(* IEC 61131-3 sources: ST_L/Practice/02_Control, 5 files *)

(* ---- 02_01_IFDemo.st ---- *)
(* ============================================================================
 * 文件: 02_01_IFDemo.st
 * 章节: 第4章 - 条件控制语句
 * 描述: IF语句完整演示
 * 学习目标: 掌握IF条件语句的各种用法
 * ============================================================================ *)

PROGRAM IFDemo
VAR
    // ==========================================================================
    // 温度监控变量
    // ==========================================================================
    iTemperature : INT := 75;      // 当前温度
    iHighLimit : INT := 100;       // 高温限值
    iLowLimit : INT := 20;         // 低温限值
    iWarningLimit : INT := 80;     // 警告限值
    bHighAlarm : BOOL;             // 高温报警
    bLowAlarm : BOOL;              // 低温报警
    bWarning : BOOL;               // 警告状态

    // ==========================================================================
    // 电机控制变量
    // ==========================================================================
    iMotorSpeed : INT := 0;
    iTargetSpeed : INT := 1500;
    bMotorRunning : BOOL := FALSE;
    bStartButton : BOOL := TRUE;
    bStopButton : BOOL := FALSE;
    bEmergencyStop : BOOL := FALSE;

    // ==========================================================================
    // 数值判断变量
    // ==========================================================================
    iScore : INT := 85;
    sGrade : STRING(2);

    iValue1, iValue2 : INT := 10;
    iMax, iMin, iMid : INT;

    // ==========================================================================
    // 边沿检测变量
    // ==========================================================================
    bCurrentInput : BOOL := FALSE;
    bLastInput : BOOL := FALSE;
    bRisingEdge : BOOL;
    iEdgeCount : INT := 0;

    // ==========================================================================
    // 数值计算变量
    // ==========================================================================
    rNumber : REAL := -3.7;
    iIntegerPart : INT;
    rFractionalPart : REAL;

    iCounter : INT := 0;
END_VAR

// ============================================================================
// 主程序逻辑
// ============================================================================
BEGIN
    // ==========================================================================
    // 1. 简单IF语句
    // ==========================================================================

    // 如果温度超过100度，触发高温报警
    IF iTemperature > iHighLimit THEN
        bHighAlarm := TRUE;
    END_IF

    // ==========================================================================
    // 2. IF-ELSE双分支
    // ==========================================================================

    // 判断电机运行状态
    IF bMotorRunning THEN
        iMotorSpeed := iTargetSpeed;
    ELSE
        iMotorSpeed := 0;
    END_IF

    // ==========================================================================
    // 3. IF-ELSIF-ELSE多分支 - 温度状态判断
    // ==========================================================================

    // 重置报警状态
    bHighAlarm := FALSE;
    bLowAlarm := FALSE;
    bWarning := FALSE;

    IF iTemperature >= iHighLimit THEN
        bHighAlarm := TRUE;
        bWarning := TRUE;
    ELSIF iTemperature <= iLowLimit THEN
        bLowAlarm := TRUE;
        bWarning := TRUE;
    ELSIF iTemperature >= iWarningLimit THEN
        bWarning := TRUE;
    ELSE
        // 温度正常
        bHighAlarm := FALSE;
        bLowAlarm := FALSE;
        bWarning := FALSE;
    END_IF

    // ==========================================================================
    // 4. IF-ELSIF-ELSE多分支 - 分数等级判定
    // ==========================================================================

    IF iScore >= 90 THEN
        sGrade := 'A';
    ELSIF iScore >= 80 THEN
        sGrade := 'B';
    ELSIF iScore >= 70 THEN
        sGrade := 'C';
    ELSIF iScore >= 60 THEN
        sGrade := 'D';
    ELSE
        sGrade := 'F';
    END_IF

    // ==========================================================================
    // 5. 嵌套IF语句 - 三角形类型判断
    // ==========================================================================
    VAR
        a, b, c : INT := 3;
        sTriangleType : STRING(20);
    END_VAR

    IF a + b > c AND b + c > a AND a + c > b THEN
        IF a = b AND b = c THEN
            sTriangleType := '等边三角形';
        ELSIF a = b OR b = c OR a = c THEN
            sTriangleType := '等腰三角形';
        ELSIF (a * a + b * b = c * c) OR (a * a + c * c = b * b) OR (b * b + c * c = a * a) THEN
            sTriangleType := '直角三角形';
        ELSE
            sTriangleType := '普通三角形';
        END_IF
    ELSE
        sTriangleType := '不能构成三角形';
    END_IF

    // ==========================================================================
    // 6. 求三个数的最大、最小、中间值
    // ==========================================================================

    iValue1 := 30;
    iValue2 := 50;

    VAR iValue3 : INT := 40; END_VAR

    IF iValue1 >= iValue2 THEN
        IF iValue1 >= iValue3 THEN
            iMax := iValue1;
            IF iValue2 >= iValue3 THEN
                iMid := iValue2;
                iMin := iValue3;
            ELSE
                iMid := iValue3;
                iMin := iValue2;
            END_IF
        ELSE
            iMax := iValue3;
            iMid := iValue1;
            iMin := iValue2;
        END_IF
    ELSE
        IF iValue2 >= iValue3 THEN
            iMax := iValue2;
            IF iValue1 >= iValue3 THEN
                iMid := iValue1;
                iMin := iValue3;
            ELSE
                iMid := iValue3;
                iMin := iValue1;
            END_IF
        ELSE
            iMax := iValue3;
            iMid := iValue2;
            iMin := iValue1;
        END_IF
    END_IF

    // ==========================================================================
    // 7. 边沿检测 - 上升沿识别
    // ==========================================================================

    bRisingEdge := bCurrentInput AND NOT bLastInput;

    IF bRisingEdge THEN
        iEdgeCount := iEdgeCount + 1;
    END_IF

    bLastInput := bCurrentInput;

    // ==========================================================================
    // 8. 浮点数处理 - 分离整数和小数部分
    // ==========================================================================

    rNumber := -3.14159;

    IF rNumber < 0.0 THEN
        iIntegerPart := REAL_TO_INT(rNumber) - 1;
    ELSE
        iIntegerPart := REAL_TO_INT(rNumber);
    END_IF

    rFractionalPart := rNumber - INT_TO_REAL(iIntegerPart);

    // ==========================================================================
    // 9. 电机启停控制（综合示例）
    // ==========================================================================

    // 急停优先级最高
    IF bEmergencyStop THEN
        bMotorRunning := FALSE;
        iMotorSpeed := 0;
    ELSIF bStopButton THEN
        bMotorRunning := FALSE;
        iMotorSpeed := 0;
    ELSIF bStartButton THEN
        bMotorRunning := TRUE;
        iMotorSpeed := iTargetSpeed;
    END_IF

    // ==========================================================================
    // 10. 计数器限幅
    // ==========================================================================

    iCounter := iCounter + 1;

    IF iCounter > 1000 THEN
        iCounter := 0;
    END_IF

END_PROGRAM

(* ---- 02_02_CASEDemo.st ---- *)
(* ============================================================================
 * 文件: 02_02_CASEDemo.st
 * 章节: 第4章 - 条件控制语句
 * 描述: CASE语句完整演示
 * 学习目标: 掌握CASE选择语句的各种用法
 * ============================================================================ *)

PROGRAM CASEDemo
VAR
    // ==========================================================================
    // 状态机变量
    // ==========================================================================
    iState : INT := 0;
    sStateName : STRING(30);

    // ==========================================================================
    // 月份处理变量
    // ==========================================================================
    iMonth : INT := 3;
    iDays : INT;
    sMonthName : STRING(20);

    // ==========================================================================
    // 菜单选择变量
    // ==========================================================================
    iMenuSelection : INT := 2;
    bExecute : BOOL := TRUE;

    // ==========================================================================
    // 报警级别变量
    // ==========================================================================
    iAlarmLevel : INT := 2;
    sAlarmMessage : STRING(50);
    bAlarmActive : BOOL := TRUE;

    // ==========================================================================
    // 枚举定义（需要定义在TYPE区域，这里用INT模拟）
    // ==========================================================================
    // MachineState: 0=IDLE, 1=STARTING, 2=RUNNING, 3=STOPPING, 4=FAULT
    iMachineState : INT := 0;

    // ==========================================================================
    // 数值范围变量
    // ==========================================================================
    iScore : INT := 78;
    iGradeLevel : INT;

    // ==========================================================================
    // 命令处理变量
    // ==========================================================================
    iCommand : INT := 16#05;
    bSuccess : BOOL;

    // ==========================================================================
    // 临时变量
    // ==========================================================================
    i : INT;
END_VAR

// ============================================================================
// 主程序逻辑
// ============================================================================
BEGIN
    // ==========================================================================
    // 1. 简单CASE语句 - 状态名称显示
    // ==========================================================================

    iState := 2;  // 假设当前状态为2

    CASE iState OF
        0:  sStateName := '初始化';
        1:  sStateName := '就绪';
        2:  sStateName := '运行中';
        3:  sStateName := '暂停';
        4:  sStateName := '停止';
        5:  sStateName := '故障';
    ELSE
        sStateName := '未知状态';
    END_CASE

    // ==========================================================================
    // 2. CASE语句 - 月份天数判断
    // ==========================================================================

    iMonth := 2;  // 2月

    CASE iMonth OF
        1, 3, 5, 7, 8, 10, 12:   // 大月
            iDays := 31;
        4, 6, 9, 11:               // 小月
            iDays := 30;
        2:                          // 2月
            iDays := 28;           // 假设非闰年
    ELSE
        iDays := 0;
    END_CASE

    // ==========================================================================
    // 3. CASE语句 - 月份名称
    // ==========================================================================

    CASE iMonth OF
        1:  sMonthName := '一月';
        2:  sMonthName := '二月';
        3:  sMonthName := '三月';
        4:  sMonthName := '四月';
        5:  sMonthName := '五月';
        6:  sMonthName := '六月';
        7:  sMonthName := '七月';
        8:  sMonthName := '八月';
        9:  sMonthName := '九月';
        10: sMonthName := '十月';
        11: sMonthName := '十一月';
        12: sMonthName := '十二月';
    ELSE
        sMonthName := '无效月份';
    END_CASE

    // ==========================================================================
    // 4. CASE语句 - 报警级别处理
    // ==========================================================================

    CASE iAlarmLevel OF
        0:  // 信息
            sAlarmMessage := '系统信息';
        1:  // 警告
            sAlarmMessage := '系统警告';
            bAlarmActive := TRUE;
        2:  // 错误
            sAlarmMessage := '系统错误';
            bAlarmActive := TRUE;
        3:  // 严重
            sAlarmMessage := '严重故障！';
            bAlarmActive := TRUE;
    ELSE
        sAlarmMessage := '未知级别';
    END_CASE

    // ==========================================================================
    // 5. CASE语句 - 分数等级判定（范围）
    // ==========================================================================

    iScore := 85;

    CASE iScore OF
        90..100:  iGradeLevel := 1;   // 优秀
        80..89:   iGradeLevel := 2;   // 良好
        70..79:   iGradeLevel := 3;   // 中等
        60..69:   iGradeLevel := 4;   // 及格
        0..59:    iGradeLevel := 5;   // 不及格
    ELSE
        iGradeLevel := 0;
    END_CASE

    // ==========================================================================
    // 6. CASE语句 - 命令解析
    // ==========================================================================

    iCommand := 3;

    CASE iCommand OF
        1:  // 启动命令
            bMotorRunning := TRUE;
            bSuccess := TRUE;
        2:  // 停止命令
            bMotorRunning := FALSE;
            bSuccess := TRUE;
        3:  // 复位命令
            iAlarmLevel := 0;
            bSuccess := TRUE;
        4:  // 急停命令
            bMotorRunning := FALSE;
            iAlarmLevel := 3;
            bSuccess := TRUE;
    ELSE
        bSuccess := FALSE;
    END_CASE

    // ==========================================================================
    // 7. CASE语句 - 菜单选择处理
    // ==========================================================================

    IF bExecute THEN
        CASE iMenuSelection OF
            1:  // 文件操作
                sStateName := '执行文件操作';
            2:  // 编辑操作
                sStateName := '执行编辑操作';
            3:  // 视图操作
                sStateName := '执行视图操作';
            4:  // 帮助
                sStateName := '显示帮助信息';
        ELSE
            sStateName := '无效菜单选择';
        END_CASE
    END_IF

    // ==========================================================================
    // 8. CASE语句 - 机器状态机
    // ==========================================================================

    CASE iMachineState OF
        0:  (* IDLE - 空闲状态 *)
            bMotorRunning := FALSE;
            iMotorSpeed := 0;
            (* 等待启动命令 *)
            IF bStartButton THEN
                iMachineState := 1;  (* 转到启动状态 *)
            END_IF

        1:  (* STARTING - 启动中 *)
            iMotorSpeed := iMotorSpeed + 100;
            IF iMotorSpeed >= iTargetSpeed THEN
                iMotorSpeed := iTargetSpeed;
                iMachineState := 2;  (* 转到运行状态 *)
            END_IF

        2:  (* RUNNING - 运行中 *)
            bMotorRunning := TRUE;
            (* 检查停止或故障 *)
            IF bStopButton THEN
                iMachineState := 3;  (* 转到停止状态 *)
            ELSIF iTemperature > 100 THEN
                iMachineState := 4;  (* 转到故障状态 *)
            END_IF

        3:  (* STOPPING - 停止中 *)
            iMotorSpeed := iMotorSpeed - 100;
            IF iMotorSpeed <= 0 THEN
                iMotorSpeed := 0;
                bMotorRunning := FALSE;
                iMachineState := 0;  (* 返回空闲状态 *)
            END_IF

        4:  (* FAULT - 故障状态 *)
            bMotorRunning := FALSE;
            iMotorSpeed := 0;
            (* 等待复位 *)
            IF bEmergencyStop THEN
                iMachineState := 0;  (* 复位后返回空闲 *)
            END_IF
    ELSE
        iMachineState := 0;  (* 默认返回空闲 *)
    END_CASE

    // ==========================================================================
    // 9. CASE语句 - 位字段解析
    // ==========================================================================
    VAR
        wControl : WORD := 16#0005;
        bBit0, bBit1, bBit2, bBit3 : BOOL;
    END_VAR

    // 解析控制字
    bBit0 := (wControl AND 16#0001) <> 0;
    bBit1 := (wControl AND 16#0002) <> 0;
    bBit2 := (wControl AND 16#0004) <> 0;
    bBit3 := (wControl AND 16#0008) <> 0;

    // 根据位字段值执行不同操作
    CASE 0 OF
        0: IF bBit0 THEN sAlarmMessage := '启用功能A'; END_IF
        1: IF bBit1 THEN sAlarmMessage := '启用功能B'; END_IF
        2: IF bBit2 THEN sAlarmMessage := '启用功能C'; END_IF
        3: IF bBit3 THEN sAlarmMessage := '启用功能D'; END_IF
    END_CASE

END_PROGRAM

(* ---- 02_03_FORDemo.st ---- *)
(* ============================================================================
 * 文件: 02_03_FORDemo.st
 * 章节: 第5章 - 循环控制语句
 * 描述: FOR循环完整演示
 * 学习目标: 掌握FOR循环的各种用法
 * ============================================================================ *)

PROGRAM FORDemo
VAR
    // ==========================================================================
    // 数组操作变量
    // ==========================================================================
    aiData : ARRAY[1..10] OF INT := [5, 2, 8, 1, 9, 3, 7, 4, 6, 10];
    aiTemperatures : ARRAY[1..24] OF INT;
    i : INT;
    iSum : DINT;
    iMax, iMin : INT;
    iMaxIndex, iMinIndex : INT;

    // ==========================================================================
    // 数学计算变量
    // ==========================================================================
    iFactorial : DINT;
    iFibonacci : DINT;
    iN : INT := 10;
    rPiApprox : REAL;
    rEApprox : REAL;

    // ==========================================================================
    // 多维数组变量
    // ==========================================================================
    amMatrix : ARRAY[1..3, 1..3] OF INT;
    amResult : ARRAY[1..3, 1..3] OF INT;

    // ==========================================================================
    // 搜索变量
    // ==========================================================================
    iTarget : INT := 7;
    bFound : BOOL := FALSE;
    iFoundIndex : INT := 0;

    // ==========================================================================
    // 临时变量
    // ==========================================================================
    rTemp : REAL;
    j, k : INT;
END_VAR

// ============================================================================
// 主程序逻辑
// ============================================================================
BEGIN
    // ==========================================================================
    // 1. 简单FOR循环 - 计算1+2+3+...+100
    // ==========================================================================

    iSum := 0;
    FOR i := 1 TO 100 DO
        iSum := iSum + i;
    END_FOR
    // iSum = 5050

    // ==========================================================================
    // 2. 逆序FOR循环
    // ==========================================================================

    iSum := 0;
    FOR i := 100 TO 1 BY -1 DO
        iSum := iSum + i;
    END_FOR
    // iSum = 5050

    // ==========================================================================
    // 3. 步长为2的FOR循环 - 计算偶数和
    // ==========================================================================

    iSum := 0;
    FOR i := 2 TO 100 BY 2 DO
        iSum := iSum + i;
    END_FOR
    // iSum = 2550

    // ==========================================================================
    // 4. 数组求和
    // ==========================================================================

    iSum := 0;
    FOR i := 1 TO 10 DO
        iSum := iSum + aiData[i];
    END_FOR
    // iSum = 55

    // ==========================================================================
    // 5. 查找最大值和最小值
    // ==========================================================================

    iMax := aiData[1];
    iMin := aiData[1];
    iMaxIndex := 1;
    iMinIndex := 1;

    FOR i := 2 TO 10 DO
        IF aiData[i] > iMax THEN
            iMax := aiData[i];
            iMaxIndex := i;
        END_IF
        IF aiData[i] < iMin THEN
            iMin := aiData[i];
            iMinIndex := i;
        END_IF
    END_FOR
    // iMax = 10, iMaxIndex = 10
    // iMin = 1, iMinIndex = 4

    // ==========================================================================
    // 6. 搜索数组中特定值
    // ==========================================================================

    bFound := FALSE;
    iFoundIndex := 0;

    FOR i := 1 TO 10 DO
        IF aiData[i] = iTarget THEN
            bFound := TRUE;
            iFoundIndex := i;
            EXIT;  (* 找到后提前退出 *)
        END_IF
    END_FOR
    // bFound = TRUE, iFoundIndex = 7

    // ==========================================================================
    // 7. 计算阶乘
    // ==========================================================================

    iN := 10;
    iFactorial := 1;
    FOR i := 1 TO iN DO
        iFactorial := iFactorial * INT_TO_DINT(i);
    END_FOR
    // iFactorial = 3628800

    // ==========================================================================
    // 8. 计算斐波那契数列
    // ==========================================================================

    iN := 10;
    VAR aiFib : ARRAY[1..20] OF DINT; END_VAR

    aiFib[1] := 1;
    aiFib[2] := 1;

    FOR i := 3 TO iN DO
        aiFib[i] := aiFib[i-1] + aiFib[i-2];
    END_FOR
    // aiFib[10] = 55

    // ==========================================================================
    // 9. 计算圆周率（莱布尼茨公式）
    // ==========================================================================

    rPiApprox := 0.0;
    FOR i := 0 TO 1000 DO
        IF (i MOD 2) = 0 THEN
            rPiApprox := rPiApprox + 4.0 / INT_TO_REAL(2 * i + 1);
        ELSE
            rPiApprox := rPiApprox - 4.0 / INT_TO_REAL(2 * i + 1);
        END_IF
    END_FOR
    // rPiApprox ≈ 3.14159

    // ==========================================================================
    // 10. 嵌套FOR循环 - 矩阵初始化
    // ==========================================================================

    FOR i := 1 TO 3 DO
        FOR j := 1 TO 3 DO
            amMatrix[i, j] := i * 10 + j;
        END_FOR
    END_FOR
    // amMatrix = [[11, 12, 13], [21, 22, 23], [31, 32, 33]]

    // ==========================================================================
    // 11. 嵌套FOR循环 - 矩阵加法
    // ==========================================================================

    FOR i := 1 TO 3 DO
        FOR j := 1 TO 3 DO
            amResult[i, j] := amMatrix[i, j] + amMatrix[i, j];
        END_FOR
    END_FOR
    // amResult = [[22, 24, 26], [42, 44, 46], [62, 64, 66]]

    // ==========================================================================
    // 12. 生成24小时温度数据（模拟）
    // ==========================================================================

    FOR i := 1 TO 24 DO
        // 模拟温度：凌晨低，中午高
        IF i <= 6 THEN
            aiTemperatures[i] := 15 + i;
        ELSIF i <= 12 THEN
            aiTemperatures[i] := 20 + (i - 6);
        ELSIF i <= 18 THEN
            aiTemperatures[i] := 28 - (i - 12);
        ELSE
            aiTemperatures[i] := 22 - (i - 18);
        END_IF
    END_FOR

    // ==========================================================================
    // 13. 条件累加 - 只累加正数
    // ==========================================================================

    iSum := 0;
    FOR i := 1 TO 10 DO
        IF aiData[i] > 0 THEN
            iSum := iSum + aiData[i];
        END_IF
    END_FOR

    // ==========================================================================
    // 14. 跳过特定值 - CONTINUE用法
    // ==========================================================================

    iSum := 0;
    FOR i := 1 TO 10 DO
        IF aiData[i] = 5 THEN
            CONTINUE;  (* 跳过值5 *)
        END_IF
        iSum := iSum + aiData[i];
    END_FOR
    // iSum = 50 (跳过了一个5)

    // ==========================================================================
    // 15. 计算数组平均值和标准差
    // ==========================================================================

    VAR
        rMean : REAL;
        rVariance : REAL;
        rStdDev : REAL;
        aiSample : ARRAY[1..10] OF INT := [10, 12, 23, 23, 16, 23, 21, 16, 18, 22];
    END_VAR

    (* 计算平均值 *)
    iSum := 0;
    FOR i := 1 TO 10 DO
        iSum := iSum + aiSample[i];
    END_FOR
    rMean := DINT_TO_REAL(iSum) / 10.0;

    (* 计算方差 *)
    rVariance := 0.0;
    FOR i := 1 TO 10 DO
        rTemp := INT_TO_REAL(aiSample[i]) - rMean;
        rVariance := rVariance + rTemp * rTemp;
    END_FOR
    rVariance := rVariance / 10.0;

    (* 计算标准差 *)
    rStdDev := SQRT(rVariance);

END_PROGRAM

(* ---- 02_04_WHILEDemo.st ---- *)
(* ============================================================================
 * 文件: 02_04_WHILEDemo.st
 * 章节: 第5章 - 循环控制语句
 * 描述: WHILE和REPEAT循环演示
 * 学习目标: 掌握条件循环的用法
 * ============================================================================ *)

PROGRAM WHILEDemo
VAR
    // ==========================================================================
    // WHILE循环变量
    // ==========================================================================
    iCounter : INT;
    iSum : INT;
    iTarget : INT := 100;
    bRunning : BOOL := TRUE;

    // ==========================================================================
    // 链表模拟变量
    // ==========================================================================
TYPE
    Node : STRUCT
        value : INT;
        next : INT;  (* 下一个节点索引，0表示无 *)
    END_STRUCT
END_TYPE

VAR
    atNodes : ARRAY[1..10] OF Node;
    iCurrent : INT;
    iListSum : INT;
    iNodeCount : INT;

    // ==========================================================================
    // 查找变量
    // ==========================================================================
    aiSortedData : ARRAY[1..20] OF INT := [1, 3, 5, 7, 9, 11, 13, 15, 17, 19, 21, 23, 25, 27, 29, 31, 33, 35, 37, 39];
    iSearchTarget : INT := 21;
    iLow, iHigh, iMid : INT;
    iSearchResult : INT := 0;  (* 0表示未找到 *)
    bSearchFound : BOOL := FALSE;

    // ==========================================================================
    // REPEAT循环变量
    // ==========================================================================
    iX : INT;
    iRepeatSum : INT;

    // ==========================================================================
    // 数据处理变量
    // ==========================================================================
    iValue : INT := 1;
    aiProcessedData : ARRAY[1..100] OF INT;
    iProcessedCount : INT := 0;
    iProcessLimit : INT := 50;

    // ==========================================================================
    // 模拟传感器变量
    // ==========================================================================
    iSensorReading : INT := 0;
    iStableReading : INT := 0;
    iStabilityCount : INT := 0;
    iLastReading : INT;
    bStable : BOOL := FALSE;

    // ==========================================================================
    // 临时变量
    // ==========================================================================
    i : INT;
END_VAR

// ============================================================================
// 主程序逻辑
// ============================================================================
BEGIN
    // ==========================================================================
    // 1. 简单WHILE循环 - 计算1+2+3+...+n直到和超过目标
    // ==========================================================================

    iCounter := 0;
    iSum := 0;

    WHILE iSum < iTarget DO
        iCounter := iCounter + 1;
        iSum := iSum + iCounter;
    END_WHILE
    // iSum >= 100, iCounter = 14 (1+2+...+14 = 105)

    // ==========================================================================
    // 2. WHILE循环 - 计算阶乘直到结果溢出
    // ==========================================================================

    iValue := 1;
    iCounter := 1;

    WHILE iValue < 1000000 AND iCounter <= 20 DO
        iCounter := iCounter + 1;
        iValue := iValue * iCounter;
    END_WHILE
    // iValue会接近但不超过1,000,000

    // ==========================================================================
    // 3. WHILE循环 - 遍历链表
    // ==========================================================================

    (* 初始化链表: 10 -> 20 -> 30 -> 0 *)
    atNodes[1].value := 10; atNodes[1].next := 2;
    atNodes[2].value := 20; atNodes[2].next := 3;
    atNodes[3].value := 30; atNodes[3].next := 0;

    iCurrent := 1;
    iListSum := 0;
    iNodeCount := 0;

    WHILE iCurrent <> 0 DO
        iListSum := iListSum + atNodes[iCurrent].value;
        iNodeCount := iNodeCount + 1;
        iCurrent := atNodes[iCurrent].next;
    END_WHILE
    // iListSum = 60, iNodeCount = 3

    // ==========================================================================
    // 4. 二分查找（使用WHILE循环）
    // ==========================================================================

    iLow := 1;
    iHigh := 20;
    bSearchFound := FALSE;

    WHILE iLow <= iHigh AND NOT bSearchFound DO
        iMid := (iLow + iHigh) / 2;

        IF aiSortedData[iMid] = iSearchTarget THEN
            bSearchFound := TRUE;
            iSearchResult := iMid;
        ELSIF aiSortedData[iMid] < iSearchTarget THEN
            iLow := iMid + 1;
        ELSE
            iHigh := iMid - 1;
        END_IF
    END_WHILE
    // iSearchResult = 11 (值21在第11个位置)

    // ==========================================================================
    // 5. REPEAT循环 - 至少执行一次
    // ==========================================================================

    iX := 100;
    iRepeatSum := 0;

    REPEAT
        iRepeatSum := iRepeatSum + iX;
        iX := iX - 1;
    UNTIL iX < 95
    END_REPEAT
    // iRepeatSum = 100+99+98+97+96 = 490

    // ==========================================================================
    // 6. WHILE vs REPEAT对比
    // ==========================================================================

    VAR
        iWhileTest, iRepeatTest : INT;
    END_VAR

    (* WHILE: 条件初始为FALSE，循环不执行 *)
    iWhileTest := 10;
    WHILE iWhileTest < 5 DO
        iWhileTest := iWhileTest + 1;
    END_WHILE
    // iWhileTest = 10 (未进入循环)

    (* REPEAT: 至少执行一次 *)
    iRepeatTest := 10;
    REPEAT
        iRepeatTest := iRepeatTest + 1;
    UNTIL iRepeatTest >= 5
    END_REPEAT
    // iRepeatTest = 11 (执行了一次)

    // ==========================================================================
    // 7. 数据处理循环
    // ==========================================================================

    iValue := 1;
    iProcessedCount := 0;

    WHILE iProcessedCount < iProcessLimit AND iValue <= 1000 DO
        iProcessedCount := iProcessedCount + 1;
        aiProcessedData[iProcessedCount] := iValue;
        iValue := iValue * 2;  (* 每次翻倍 *)
    END_WHILE
    // 处理了直到2^5 = 32的所有值

    // ==========================================================================
    // 8. 传感器稳定性检测
    // ==========================================================================

    iStabilityCount := 0;
    iLastReading := iSensorReading;

    WHILE iStabilityCount < 5 AND NOT bStable DO
        iSensorReading := iSensorReading + 1;  (* 模拟读取 *)
        (* 实际应用中这里应该是真实的传感器读取 *)

        IF ABS(iSensorReading - iLastReading) <= 2 THEN
            iStabilityCount := iStabilityCount + 1;
        ELSE
            iStabilityCount := 0;
        END_IF

        iLastReading := iSensorReading;

        IF iStabilityCount >= 5 THEN
            bStable := TRUE;
            iStableReading := iSensorReading;
        END_IF
    END_WHILE

    // ==========================================================================
    // 9. 最大公约数（欧几里得算法）
    // ==========================================================================

    VAR
        iGCD_A, iGCD_B, iTemp : INT;
    END_VAR

    iGCD_A := 48;
    iGCD_B := 18;

    WHILE iGCD_B <> 0 DO
        iTemp := iGCD_B;
        iGCD_B := iGCD_A MOD iGCD_B;
        iGCD_A := iTemp;
    END_WHILE
    // iGCD_A = 6 (48和18的最大公约数)

    // ==========================================================================
    // 10. 嵌套循环 - 质数判断
    // ==========================================================================

    VAR
        iPrimeTest : INT := 97;
        iDivisor : INT;
        bIsPrime : BOOL := TRUE;
    END_VAR

    iDivisor := 2;

    WHILE iDivisor * iDivisor <= iPrimeTest AND bIsPrime DO
        IF iPrimeTest MOD iDivisor = 0 THEN
            bIsPrime := FALSE;
        END_IF
        iDivisor := iDivisor + 1;
    END_WHILE
    // bIsPrime = TRUE (97是质数)

    // ==========================================================================
    // 11. 生成斐波那契数列直到超过阈值
    // ==========================================================================

    VAR
        aiFib : ARRAY[1..30] OF DINT;
        iFibCount : INT := 2;
    END_VAR

    aiFib[1] := 1;
    aiFib[2] := 1;

    WHILE aiFib[iFibCount] < 1000 DO
        iFibCount := iFibCount + 1;
        aiFib[iFibCount] := aiFib[iFibCount-1] + aiFib[iFibCount-2];
    END_WHILE
    // iFibCount = 16, aiFib[16] = 987 (< 1000)
    // 下一个是1597 (> 1000)

END_PROGRAM

(* ---- 02_05_MotorControl.st ---- *)
(* ============================================================================
 * 文件: 02_05_MotorControl.st
 * 章节: 第5章 - 综合练习
 * 描述: 电机控制系统 - 综合运用条件与循环语句
 * 学习目标: 综合运用IF、CASE、FOR循环解决实际问题
 * ============================================================================ *)

PROGRAM MotorControl
VAR
    // ==========================================================================
    // 输入变量
    // ==========================================================================
    bStartButton AT %IX0.0 : BOOL;      // 启动按钮
    bStopButton AT %IX0.1 : BOOL;       // 停止按钮
    bResetButton AT %IX0.2 : BOOL;      // 复位按钮
    bEmergencyStop AT %IX0.3 : BOOL;    // 急停
    bHomeSensor AT %IX1.0 : BOOL;       // 原点传感器
    bLimitSwitch AT %IX1.1 : BOOL;      // 限位开关
    iTargetPosition AT %IW0 : INT;      // 目标位置

    // ==========================================================================
    // 输出变量
    // ==========================================================================
    bMotorRun AT %QX0.0 : BOOL;        // 电机运行
    bMotorDirection AT %QX0.1 : BOOL;   // 电机方向 (0=正转,1=反转)
    bBrake AT %QX0.2 : BOOL;            // 制动器
    bIndicator AT %QX1.0 : BOOL;        // 指示灯
    iMotorSpeed AT %QW0 : INT;         // 电机速度
    iCurrentPosition AT %QW1 : INT;    // 当前位置

    // ==========================================================================
    // 内部变量
    // ==========================================================================
    iState : INT := 0;                  // 状态机状态
    iSpeedProfile : ARRAY[1..5] OF INT := [100, 500, 1000, 1500, 2000];  // 速度曲线
    iCurrentStage : INT := 1;           // 当前加速阶段
    iTimer : INT := 0;                  // 定时器
    iCycleCount : INT := 0;             // 循环计数
    iErrorCode : INT := 0;              // 错误代码

    // 边沿检测
    bLastStart : BOOL := FALSE;
    bLastStop : BOOL := FALSE;
    bLastReset : BOOL := FALSE;

    // 数据记录
    aiSpeedHistory : ARRAY[1..100] OF INT;
    iHistoryIndex : INT := 1;
END_VAR

// ============================================================================
// 状态定义
// ============================================================================
// 0 = STOPPED    - 停止
// 1 = STARTING   - 启动中
// 2 = ACCEL      - 加速中
// 3 = RUNNING    - 运行中
// 4 = DECEL      - 减速中
// 5 = HOMING     - 回原中
// 9 = FAULT      - 故障

// ============================================================================
// 错误代码定义
// ============================================================================
// 0 = 无错误
// 1 = 急停触发
// 2 = 限位触发
// 3 = 过温
// 4 = 过流

// ============================================================================
// 主程序逻辑
// ============================================================================
BEGIN
    // ==========================================================================
    // 1. 边沿检测
    // ==========================================================================
    VAR
        bStartEdge : BOOL;
        bStopEdge : BOOL;
        bResetEdge : BOOL;
    END_VAR

    bStartEdge := bStartButton AND NOT bLastStart;
    bStopEdge := bStopButton AND NOT bLastStop;
    bResetEdge := bResetButton AND NOT bLastReset;

    bLastStart := bStartButton;
    bLastStop := bStopButton;
    bLastReset := bResetButton;

    // ==========================================================================
    // 2. 急停处理（最高优先级）
    // ==========================================================================

    IF bEmergencyStop THEN
        iState := 9;                    // 故障状态
        iErrorCode := 1;
        bMotorRun := FALSE;
        bBrake := TRUE;
        iMotorSpeed := 0;
        bIndicator := FALSE;
    END_IF

    // ==========================================================================
    // 3. 主状态机
    // ==========================================================================

    CASE iState OF
        // --------------------------------------------------------------------------
        // 状态0: 停止
        // --------------------------------------------------------------------------
        0:
            bMotorRun := FALSE;
            bBrake := TRUE;
            iMotorSpeed := 0;
            iCurrentStage := 1;

            IF bStartEdge THEN
                IF NOT bHomeSensor THEN
                    // 需要回原
                    iState := 5;
                ELSE
                    // 直接启动
                    iState := 1;
                END_IF
            END_IF

        // --------------------------------------------------------------------------
        // 状态1: 启动中
        // --------------------------------------------------------------------------
        1:
            bBrake := FALSE;
            bMotorRun := TRUE;
            iMotorSpeed := iSpeedProfile[1];
            iTimer := 0;
            iState := 2;  // 自动转入加速

        // --------------------------------------------------------------------------
        // 状态2: 加速中
        // --------------------------------------------------------------------------
        2:
            iTimer := iTimer + 1;

            IF iTimer >= 100 THEN  // 每100ms加速一次
                iTimer := 0;
                iCurrentStage := iCurrentStage + 1;

                IF iCurrentStage <= 5 THEN
                    iMotorSpeed := iSpeedProfile[iCurrentStage];
                ELSE
                    iState := 3;  // 达到目标速度
                END_IF
            END_IF

            // 检查限位
            IF bLimitSwitch THEN
                iState := 9;
                iErrorCode := 2;
            END_IF

        // --------------------------------------------------------------------------
        // 状态3: 运行中
        // --------------------------------------------------------------------------
        3:
            iMotorSpeed := iSpeedProfile[5];  // 全速运行

            // 位置控制
            IF iCurrentPosition < iTargetPosition THEN
                bMotorDirection := FALSE;  // 正转
            ELSIF iCurrentPosition > iTargetPosition THEN
                bMotorDirection := TRUE;   // 反转
            END_IF

            // 接近目标时减速
            IF ABS(iCurrentPosition - iTargetPosition) < 100 THEN
                iState := 4;
                iCurrentStage := 5;
                iTimer := 0;
            END_IF

            // 检查限位
            IF bLimitSwitch THEN
                iState := 9;
                iErrorCode := 2;
            END_IF

            // 停止命令
            IF bStopEdge THEN
                iState := 4;
                iCurrentStage := 5;
                iTimer := 0;
            END_IF

            // 指示灯闪烁
            bIndicator := (iCycleCount < 50);
            iCycleCount := iCycleCount + 1;
            IF iCycleCount >= 100 THEN
                iCycleCount := 0;
            END_IF

        // --------------------------------------------------------------------------
        // 状态4: 减速中
        // --------------------------------------------------------------------------
        4:
            iTimer := iTimer + 1;

            IF iTimer >= 100 THEN
                iTimer := 0;
                iCurrentStage := iCurrentStage - 1;

                IF iCurrentStage >= 1 THEN
                    iMotorSpeed := iSpeedProfile[iCurrentStage];
                END_IF

                IF iCurrentStage <= 1 THEN
                    iState := 0;  // 停止
                END_IF
            END_IF

        // --------------------------------------------------------------------------
        // 状态5: 回原中
        // --------------------------------------------------------------------------
        5:
            bMotorDirection := TRUE;  // 反转
            bMotorRun := TRUE;
            bBrake := FALSE;
            iMotorSpeed := iSpeedProfile[2];

            IF bHomeSensor THEN
                iCurrentPosition := 0;
                bMotorRun := FALSE;
                bBrake := TRUE;
                iState := 1;  // 回到启动流程
            END_IF

        // --------------------------------------------------------------------------
        // 状态9: 故障
        // --------------------------------------------------------------------------
        9:
            bMotorRun := FALSE;
            bBrake := TRUE;
            iMotorSpeed := 0;
            bIndicator := TRUE;  // 故障指示灯亮

            IF bResetEdge THEN
                iErrorCode := 0;
                iState := 0;
                bIndicator := FALSE;
            END_IF

    ELSE
        iState := 0;
    END_CASE

    // ==========================================================================
    // 4. 模拟位置变化（实际应用中由编码器反馈）
    // ==========================================================================

    IF bMotorRun THEN
        IF bMotorDirection THEN
            iCurrentPosition := iCurrentPosition - (iMotorSpeed / 100);
        ELSE
            iCurrentPosition := iCurrentPosition + (iMotorSpeed / 100);
        END_IF
    END_IF

    // ==========================================================================
    // 5. 速度历史记录
    // ==========================================================================

    iHistoryIndex := (iHistoryIndex MOD 100) + 1;
    aiSpeedHistory[iHistoryIndex] := iMotorSpeed;

    // ==========================================================================
    // 6. 错误代码显示（通过指示灯闪烁次数表示）
    // ==========================================================================

    IF iState = 9 THEN
        VAR iBlinkCount : INT := 0; END_VAR
        iBlinkCount := 0;
        // 闪烁iErrorCode次
    END_IF

END_PROGRAM
